GLOBALCONSTANTS DataPanel_MI_DO (* DataPanel Modules with medium IO density DO constants *)
  (* Standard: 61499-1; Description: Copyright (c) 2024 HR Agrartechnik GmbH This program and the accompanying materials are made available under the terms of the Eclipse Public License 2.0 which is available at https://www.eclipse.org/legal/epl-2.0/ SPDX-License-Identifier: EPL-2.0 *)
  (* Version 1.0, 2024-01-25, Franz Höpfinger, HR Agrartechnik GmbH *)
  VAR_GLOBAL CONSTANT
    Output_Q1 : DataPanel_MI_DO_S := (Pin := 1);
    Output_Q2 : DataPanel_MI_DO_S := (Pin := 2);
    Output_Q3 : DataPanel_MI_DO_S := (Pin := 3);
    Output_Q4 : DataPanel_MI_DO_S := (Pin := 4);
    Output_Q5 : DataPanel_MI_DO_S := (Pin := 5);
    Output_Q6 : DataPanel_MI_DO_S := (Pin := 6);
    Output_Q7 : DataPanel_MI_DO_S := (Pin := 7);
    Output_Q8 : DataPanel_MI_DO_S := (Pin := 8);
    Output_Q9 : DataPanel_MI_DO_S := (Pin := 9);
    Invalid : DataPanel_MI_DO_S := (Pin := 255);
  END_VAR
END_GLOBALCONSTANTS
